TYPE DMX_Control :
STRUCT
	TransmitRequest : BIT;
	DisableCyclicTxD : BIT;
	SendDefaultData : BIT;
	ChannelLength : UINT;
	StartCode : USINT;
END_STRUCT
END_TYPE

(* stored: Version 1.1.0.1
   DUT DMX_Control: Id {44b57fa9-0c17-449d-87e7-1caecb8b895b} *)
